(* CODESYS project building automation test.project

Project tree, tasks and I/O mapping:
  Device : L-force Controller c300 Logic, Lenze, order no. LPC 1000, version 3.8.0.0
    application Application
      libraries: L_Util, 3.3.0.0 (Lenze); L_PLCDataManagerAccess, 3.0.0.0 (Lenze); L_PLCLoggingAccess, 3.3.0.0 (Lenze)
      task MainTask (cyclic, interval t#10ms, priority 1) calls PLC_PRG
      program PLC_PRG [LD]
    Coupler_I_O_moduls : Coupler I/O moduls, Lenze, version 3.6.0.0
        settings: Count groups = 1; Application Name of Task = 'Application'; Group1 Task Name = 'MainTask'
        unmapped channels: Error, unused, unused, unused, unused, unused, unused, unused, ErrorID, AbsoluteCounter, ErrorReset, unused, unused, unused, unused, unused, unused, unused
      EPM_S202 : EPM-S202: DI8, DC 24V, Lenze, order no. EPM-S202, version 3.6.0.0
          settings: Group = 0; Task Guid = '00000000-0000-0000-0000-000000000000'
          input  Application.PLC_PRG.xDoorStateLocked : BIT  // DI1
          input  Application.PLC_PRG.xdoorStateUnlocked : BIT  // DI2
          input  Application.PLC_PRG.xMasterAlarmReset : BIT  // DI3
          input  Application.PLC_PRG.xEndofDayInput : BIT  // DI4
          input  Application.PLC_PRG.xStartofDayInput : BIT  // DI5
          input  Application.PLC_PRG.xDoor_1_Open : BIT  // DI6
          input  Application.PLC_PRG.xDoorCodeInput : BIT  // DI7
          unmapped channels: DI8
      EPM_S302 : EPM-S302: DO8, DC 24V, 0.5A, Lenze, order no. EPM-S302, version 3.6.0.0
          settings: Group = 0; Task Guid = '00000000-0000-0000-0000-000000000000'
          output Application.PLC_PRG.xDoor_1_Lock : BIT  // DO1
          output Application.PLC_PRG.xset_fireLight : BIT  // DO2
          output Application.PLC_PRG.xset_fireSounder : BIT  // DO3
          output Application.PLC_PRG.xSet_falseEntryAlarm : BIT  // DO4
          output Application.PLC_PRG.xset_doorUnlockedbyCode : BIT  // DO5
          unmapped channels: DO6, DO7, DO8
*)

// Device/Application/PLC_PRG
PROGRAM PLC_PRG

VAR
	xDoorStateLocked: BOOL;
	xset_doorStateLocked: BOOL;
	xDoor_1_Lock: BOOL;
	xset_doorStateUnlocked: BOOL;
	xdoorStateUnlocked: BOOL;
	xfireAlarm: BOOL;
	xset_fireAlarm: BOOL;
	xset_fireLight: BOOL;
	xset_fireSounder: BOOL;
	xMasterAlarmReset: BOOL;
	xset_masterAlarmReset: BOOL;
	xEndofDayInput: BOOL;
	xroom216MotionSensor: BOOL;
	xset_EndofDay: BOOL;
	xSet_falseEntryAlarm: BOOL;
	xDoor_1_Open: BOOL;
	xset_EndofDayInput: BOOL;
	xStartofDayInput: BOOL;
	xset_StartofdayInput: BOOL;
	xDoorCodeInput: BOOL;
	xset_DoorCodeUnlocked: BOOL;
	xset_doorUnlockedbyCode: BOOL;
	xset_doorCodeLocked: BOOL;
	delay: TON;
	xcodeUnlockedCondition: BOOL;
	xdoorCodeHigh: BOOL;
	test: RS;
	xdoorCodeLow: BOOL;
END_VAR
VAR // added by the converter: edge detectors and wires of the graphical bodies
    _w1, _w2, _w3, _w4, _w5, _w6, _w7, _w8, _w9, _w10, _w11 : BOOL;
END_VAR

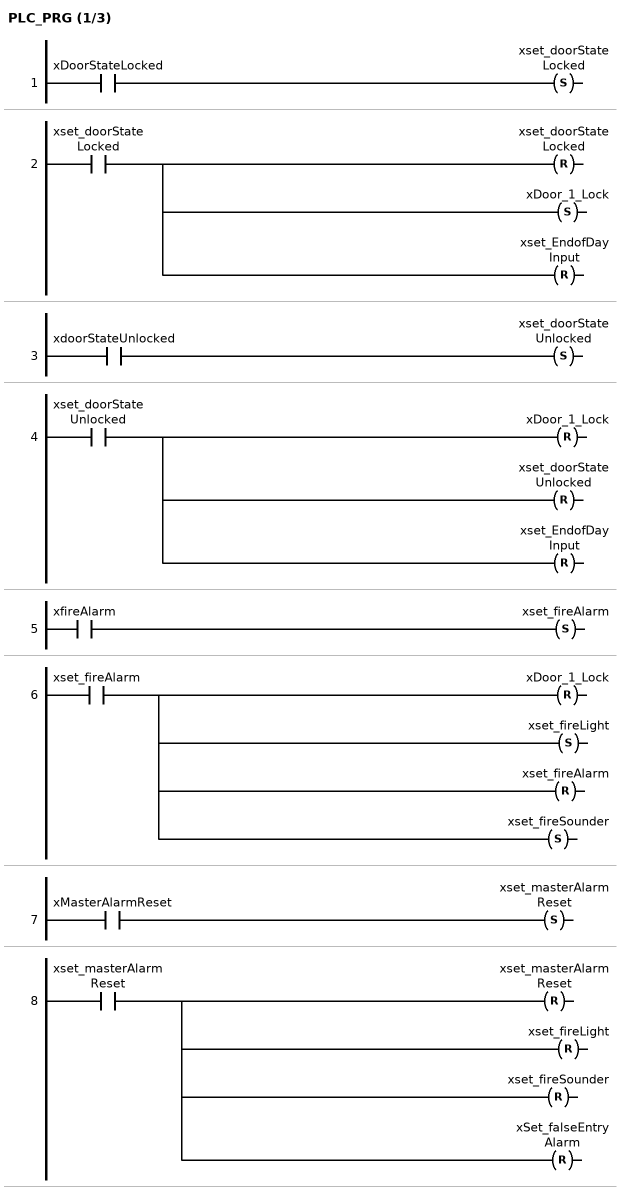
// NETWORK 1
xset_doorStateLocked S= xDoorStateLocked;

// NETWORK 2
_w1 := xset_doorStateLocked;
xset_doorStateLocked R= _w1;
xDoor_1_Lock S= _w1;
xset_EndofDayInput R= _w1;

// NETWORK 3
xset_doorStateUnlocked S= xdoorStateUnlocked;

// NETWORK 4
_w2 := xset_doorStateUnlocked;
xDoor_1_Lock R= _w2;
xset_doorStateUnlocked R= _w2;
xset_EndofDayInput R= _w2;

// NETWORK 5
xset_fireAlarm S= xfireAlarm;

// NETWORK 6
_w3 := xset_fireAlarm;
xDoor_1_Lock R= _w3;
xset_fireLight S= _w3;
xset_fireAlarm R= _w3;
xset_fireSounder S= _w3;

// NETWORK 7
xset_masterAlarmReset S= xMasterAlarmReset;

// NETWORK 8
_w4 := xset_masterAlarmReset;
xset_masterAlarmReset R= _w4;
xset_fireLight R= _w4;
xset_fireSounder R= _w4;
xSet_falseEntryAlarm R= _w4;

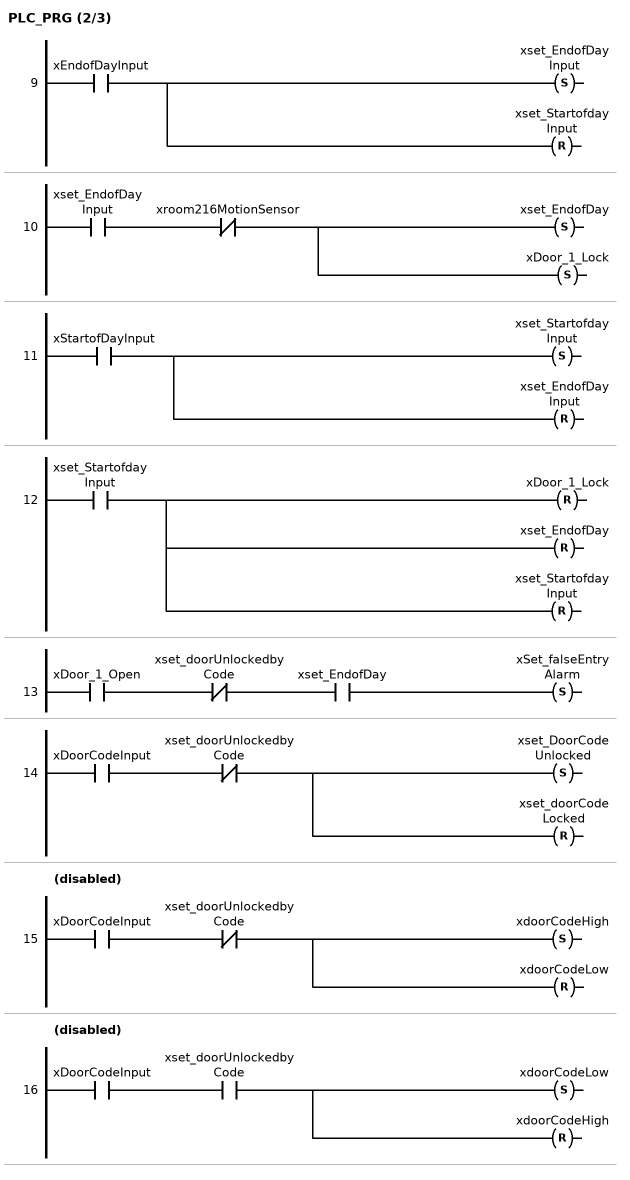
// NETWORK 9
xset_EndofDayInput S= xEndofDayInput;
xset_StartofdayInput R= xEndofDayInput;

// NETWORK 10
_w5 := xset_EndofDayInput AND NOT xroom216MotionSensor;
xset_EndofDay S= _w5;
xDoor_1_Lock S= _w5;

// NETWORK 11
xset_StartofdayInput S= xStartofDayInput;
xset_EndofDayInput R= xStartofDayInput;

// NETWORK 12
xDoor_1_Lock R= xset_StartofdayInput;
xset_EndofDay R= xset_StartofdayInput;
xset_StartofdayInput R= xset_StartofdayInput;

// NETWORK 13
xSet_falseEntryAlarm S= xDoor_1_Open AND NOT xset_doorUnlockedbyCode AND xset_EndofDay;

// NETWORK 14
_w6 := xDoorCodeInput AND NOT xset_doorUnlockedbyCode;
xset_DoorCodeUnlocked S= _w6;
xset_doorCodeLocked R= _w6;

// NETWORK 15 (disabled)
// _w7 := xDoorCodeInput AND NOT xset_doorUnlockedbyCode;
// xdoorCodeHigh S= _w7;
// xdoorCodeLow R= _w7;

// NETWORK 16 (disabled)
// _w8 := xDoorCodeInput AND xset_doorUnlockedbyCode;
// xdoorCodeLow S= _w8;
// xdoorCodeHigh R= _w8;

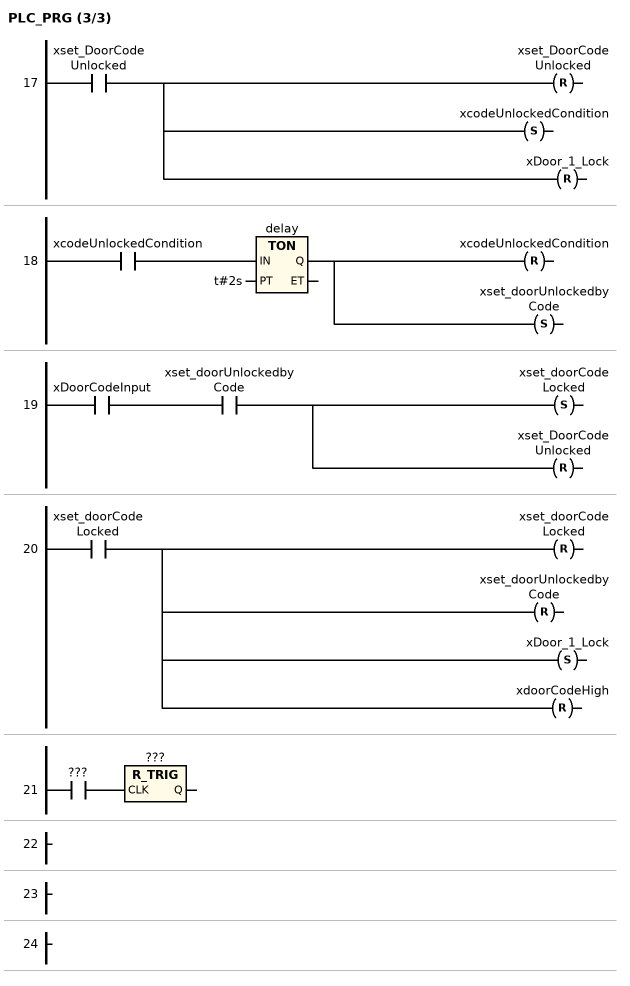
// NETWORK 17
_w9 := xset_DoorCodeUnlocked;
xset_DoorCodeUnlocked R= _w9;
xcodeUnlockedCondition S= _w9;
xDoor_1_Lock R= _w9;

// NETWORK 18
delay(IN := xcodeUnlockedCondition, PT := t#2s); // TON
xcodeUnlockedCondition R= delay.Q;
xset_doorUnlockedbyCode S= delay.Q;

// NETWORK 19
_w10 := xDoorCodeInput AND xset_doorUnlockedbyCode;
xset_doorCodeLocked S= _w10;
xset_DoorCodeUnlocked R= _w10;

// NETWORK 20
_w11 := xset_doorCodeLocked;
xset_doorCodeLocked R= _w11;
xset_doorUnlockedbyCode R= _w11;
xDoor_1_Lock S= _w11;
xdoorCodeHigh R= _w11;

// NETWORK 21
???(); // R_TRIG

// NETWORK 22

// NETWORK 23

// NETWORK 24

END_PROGRAM
